# EPICS substitutions: ek9000App/Db/EL3042.substitutions
file EL3042.template
{       pattern
        {
                TERMINAL,

        }
        {
        }
}
